{attribute 'GeneratedUsingTerminal: EP3356-0022-0016'}
{attribute addProperty BoxType "EP3356-0022-0016"}
{attribute addProperty Id "ValueAT %I*DINT4"}
{attribute addProperty CRC "3910704203"}
{attribute addProperty Size "4"}
TYPE RMB_Value_INT_E9189C4B :
STRUCT
	{attribute addProperty Name "Value"}
	Value AT %I* : DINT;
END_STRUCT
END_TYPE

(* stored: Version 1.2.0.0, ProductVersion 3.1.4024.9
   DUT RMB_Value_INT_E9189C4B: Id {c6282233-6269-48c7-ac43-a8a606559e02} *)
